// TIA Portal V17 export
// export: Created 2025-11-19T10:30:00.000Z, ExportSetting WithDefaults, DisplayName Totally Integrated Automation Portal, DisplayVersion V17
FUNCTION_BLOCK "FB_PID_Controller"   // FB20, SCL
{ S7_Optimized_Access := 'TRUE' }
AUTHOR : Control Systems
FAMILY : Controllers
NAME : PID Controller
VERSION : 2.1
// stored: AutoNumber true, IsIECCheckEnabled true
   VAR_INPUT
      Setpoint : Real;
      ProcessValue : Real;
      Kp : Real;
      Ki : Real;
      Kd : Real;
      Enable : Bool;
   END_VAR
   VAR_OUTPUT
      ControlOutput : Real;
      Error : Real;
   END_VAR
   VAR
      IntegralSum : Real;
      LastError : Real;
      Initialized : Bool;
   END_VAR
   VAR_TEMP
      PropTerm : Real;
      IntTerm : Real;
      DiffTerm : Real;
   END_VAR
BEGIN
// PID Control Algorithm
// PID controller with anti-windup protection
   // PID Controller Implementation
   IF #Enable THEN
       // Calculate error
       #Error := #Setpoint - #ProcessValue;

       // Proportional term
       #PropTerm := #Kp * #Error;

       // Integral term
       #IntegralSum := #IntegralSum + #Error;
       #IntTerm := #Ki * #IntegralSum;

       // Derivative term
       IF #Initialized THEN
           #DiffTerm := #Kd * (#Error - #LastError);
       ELSE
           #DiffTerm := 0.0;
           #Initialized := TRUE;
       END_IF;

       // Calculate control output
       #ControlOutput := #PropTerm + #IntTerm + #DiffTerm;

       // Anti-windup
       IF #ControlOutput > 100.0 THEN
           #ControlOutput := 100.0;
           #IntegralSum := #IntegralSum - #Error;
       ELSIF #ControlOutput < 0.0 THEN
           #ControlOutput := 0.0;
           #IntegralSum := #IntegralSum - #Error;
       END_IF;

       // Save error for next cycle
       #LastError := #Error;
   ELSE
       // Reset controller
       #ControlOutput := 0.0;
       #IntegralSum := 0.0;
       #LastError := 0.0;
       #Initialized := FALSE;
   END_IF;
END_FUNCTION_BLOCK
